Universal Robots URScript: dusan_v3_nosensor.task.script

def dusan_v3_nosensor():
  # Preamble Script.
  # Test Preamble Script To Be Added In The Future.
  set_safety_mode_transition_hardness(1)
  # Configuration Preamble Script.
  # Configuration variables.
  #
  global Home_joint
  Home_joint = [0.55498, -1.00739, -2.64993, -1.05507, 1.5708, 0.55497]
  #
  global Home_pose
  Home_pose = [0.33684, -0.00001, 0.31805, 3.14159, 0, -1.57079]
  # 시작 포즈 (입력레지스터 316~321). UI가 저장한 값
  global start_pose
  start_pose = [0.33684, -0.00001, 0.31805, 3.14159, 0, -1.57079]
  # 0=이 변수값 사용, 1=Modbus 310~321 사용 (레지스터 308)
  global pose_src
  pose_src = 0
  # 작업 속도 입력 [mm/s] (입력레지스터 306). 0이면 v_l 유지
  global spd_in
  spd_in = 0
  # 로봇 자체 속도 비율 [%] 2~100 (입력레지스터 307)
  global spd_ratio
  spd_ratio = 100
  # 0=이 변수값 사용, 1=Modbus 256~259 사용 (레지스터 266)
  global param_src
  param_src = 0
  # 중앙 접촉 센서 1차 — ON 이면 적정 눌림 위치
  global di_touch
  di_touch = 0
  # 중앙 접촉 센서 2차 — ON 이면 눌림 한계. TCP +Y 로 후퇴한다
  global di_limit
  di_limit = 1
  # 도면 반지름(안쪽 면) [mm]. 레지스터 260 을 0.1mm 로 받고, dus_init 이 두께를 더해 훑는 면 반지름으로 바꾼다
  global app_radius
  app_radius = 894.59998
  # 제품 두께 [mm]. 레지스터 261 을 0.1mm 단위로 받는다. UT 기록용
  global app_thick
  app_thick = 10
  # 격자 가로 = 호 길이 [mm] (레지스터 256). 로봇이 실제로 지나는 거리. 현이 아니다
  global app_arc
  app_arc = 1110
  # EOAT 가로(호 방향) [mm]. 레지스터 262. 5축 X형 257 / 8축 직사각 186
  global eoat_w
  eoat_w = 257
  # EOAT 세로 [mm]. 레지스터 263. 5축 257 / 8축 316(세로로 길게). 스캐너 밴드 높이로 쓴다
  global eoat_h
  eoat_h = 257
  # TCP 가 실제로 움직일 호 길이 [mm] = app_arc - eoat_w. dus_init 이 계산
  global arc_run
  arc_run = 853
  # 곡률 중심 X [m]. probe_l 이 계산
  global arc_ox
  arc_ox = 1.53144
  # 곡률 중심 Y [m]. probe_l 이 계산
  global arc_oy
  arc_oy = -0.00002
  # 원점(zero_pose)이 곡률 중심에서 보이는 각 [rad]
  global arc_phi0
  arc_phi0 = 2.66484
  # 호 기준이 잡혔는지. True 여야 호 위치를 발행한다
  global arc_ok
  arc_ok = True
  # 원점부터 지금까지의 호 위 거리 [mm]. 레지스터 286 으로 발행
  global arc_s
  arc_s = 0
  # 호 반각 [rad] = app_arc/(2*app_radius). dus_init 이 계산
  global arc_half
  arc_half = 0.47675
  # 센서로 잰 적정 눌림 보정량 [m]. 계산한 3점을 TCP -Y 로 이만큼 더 민다
  global press_off
  press_off = 0
  # 자세 보정 중 한 걸음 전진/후퇴 거리 [mm]
  global seek_step
  seek_step = 2
  # 전진·회전 되풀이 최대 횟수. 넘으면 포기하고 진행
  global seek_tries
  seek_tries = 80
  # 전진 최대 거리 [mm]. 센서가 없으면 여기까지 가고 멈춘다
  global seek_limit
  seek_limit = 400
  # 센서판: 계산한 좌우 끝점 접근 전 대기 거리 [mm](TCP +Y로 물러난 지점). 논센서판: 센서 없이 전진할 고정 거리 [mm]
  global probe_dist
  probe_dist = 300
  # [임시판 전용] 중앙이 가장자리보다 더 전진할 거리 [mm]. 0 이면 app_diameter 로 자동 계산(바깥 볼록면이라 음수가 나온다). 손으로 넣으려면 0 이 아닌 값을 준다
  global probe_bow
  probe_bow = 0
  # [임시판 전용] 원통 지름 [mm]. probe_bow 가 0 일 때 호의 볼록량을 이 값으로 계산한다 (센서가 붙으면 필요 없다)
  global app_diameter
  app_diameter = 1669
  # 측정 후 후퇴 거리 [mm]
  global back_off
  back_off = 100
  # 가로 패스를 나누는 구간 길이 [mm]. 작을수록 X 보정이 촘촘하다
  global seg_len
  seg_len = 50
  # movel(스캔 제외) 속도 [m/s]. dus_init 이 150mm/s 로 상한을 자른다
  global v_l
  v_l = 0.15
  # movel(스캔 제외) 가속도 [m/s^2]. 필요하면 각 스크립트가 그 자리에서 바꿔 쓴다
  global a_l
  a_l = 1.2
  # movej 속도 [rad/s] (20 deg/s). dus_init 이 0.50 rad/s 로 상한을 자른다 — 조그 상한과 같다. 펜던트 MoveJ 노드(홈 복귀)는 이 값을 직접 참조하지 못하므로 노드 쪽 수치도 같이 맞춰 둬야 한다
  global v_j
  v_j = 0.3490658503988659
  # movej 가속도 [rad/s^2] (40 deg/s^2)
  global a_j
  a_j = 0.698131700835289
  # 스캔 movel/movec 속도 [m/s]. 고정 스펙 100mm/s
  global v_scan
  v_scan = 0.1
  # 스캔 movel/movec 가속도 [m/s^2]. 고정 스펙 400mm/s^2
  global a_scan
  a_scan = 0.4
  # 작업 영역 좌우 너비 [mm] (입력레지스터 256)
  global app_width
  app_width = 821.05219
  # 작업 영역 높이 [mm] (입력레지스터 257)
  global app_height
  app_height = 500
  # 스캐너 세로 유효높이 [mm] (입력레지스터 258)
  global scan_h
  scan_h = 257
  # 세로 겹침 [mm] (입력레지스터 259)
  global overlap
  overlap = 20
  # 상승 피치 = scan_h - overlap [mm] (고정)
  global pitch
  pitch = 237
  # 가로 패스 수
  global rows
  rows = 3
  # 완료한 가로 패스 수
  global row_idx
  row_idx = 1
  # 1=오른쪽(Y-) 차례, -1=왼쪽(Y+) 차례
  global dir_sign
  dir_sign = -1
  #
  global pass_done
  pass_done = 0
  # 측정 완료한 점 수 (0~3)
  global n_probe
  n_probe = 3
  # 센서로 검출된 점 수
  global n_hit
  n_hit = 0
  # 중앙 측정 X [m]
  global p_cx
  p_cx = 0.63684
  # Y+ 끝 측정 X [m]
  global p_lx
  p_lx = 0.7366
  # Y- 끝 측정 X [m]
  global p_rx
  p_rx = 0.7366
  # 중앙 Y [m]
  global y_c
  y_c = -0.00001
  #
  global y_l
  y_l = 0.30185
  #
  global y_r
  y_r = -0.29815
  # 너비의 절반 [m]
  global half
  half = 0.3
  # 벽면 2차식 계수 : x = qa*dy^2 + qb*dy + qc, dy = Y - y_c
  global qa
  qa = 0
  # 벽면 2차식 1차항
  global qb
  qb = 0
  # 벽면 2차식 상수항 (= 중앙 X)
  global qc
  qc = 0
  #
  global zero_ok
  zero_ok = True
  #
  global x_start
  x_start = [0.33684, -0.00001, 0.32105, 3.14159, -0, -1.57079]
  #
  global z_base
  z_base = 0.32105
  # 원점 = Y+ 끝 측정 위치
  global zero_pose
  zero_pose = [0.7366, 0.41051, 0.32105, 3.14159, -0.00001, -2.04755]
  # pose_inv(zero_pose)
  global zero_inv
  zero_inv = [0.70276, 0.46608, 0.32105, -3.14159, 0, -2.04755]
  # 현재 절대 TCP (260~265 로 발행)
  global cur_pose
  cur_pose = [0.7236, -0.38435, 0.55805, 3.14159, -0.00001, -1.12675]
  # 원점 기준 상대 pose (280~285 로 발행)
  global rel_pose
  rel_pose = [-0.013, -0.79486, 0.237, -0, -0, 0.9208]
  # 현재 구간 목표 pose
  global tgt_pose
  tgt_pose = [0.7366, -0.41054, 0.55805, -3.14159, -0.00001, -1.09406]
  #
  global dy
  dy = 0.3
  #
  global y_from
  y_from = -0.30001
  #
  global y_to
  y_to = 0.29999
  #
  global n_seg
  n_seg = 12
  #
  global i_seg
  i_seg = 13
  # 누적 이동거리 [mm]
  global path_len
  path_len = 1090
  # 워치독 카운터
  global alive
  alive = 14011
  # 이동 스레드 핸들
  global mv_h
  mv_h = 0
  # 발행 스레드 핸들
  global pub_h
  pub_h = 855631424
  # 정렬 전 기준 자세. 측정점 사이를 이동할 때 여기로 되돌린다 (probe_c 가 채운다)
  global probe_rot
  probe_rot = [0.33684, -0.00001, 0.31805, 3.14159, 0, -1.57079]
  # movec 의 mode. 0 = 자세 고정
  global arc_mode
  arc_mode = 0
  # 중앙 측정 pose — movec 의 경유점 (330~335 로 발행)
  global p_c_pose
  p_c_pose = [0.63684, -0.00001, 0.32105, 3.14159, -0.00001, -1.5708]
  # Y- 끝 측정 pose — movec 의 도착점 (340~345 로 발행)
  global p_r_pose
  p_r_pose = [0.7366, -0.41054, 0.32105, 3.14159, -0.00001, -1.09405]
  # movec 경유점 (현재 높이로 갈아끼운 것)
  global via_pose
  via_pose = [0.63684, -0.00001, 0.55805, 3.14159, -0.00001, -1.5708]
  # movec 도착점 (현재 높이로 갈아끼운 것)
  global to_pose
  to_pose = [0.7366, 0.41051, 0.55805, 3.14159, -0.00001, -2.04755]
  # 가로 패스 시작 시점의 Z [m]
  global z_now
  z_now = 0.55805
  set_tool_analog_io_work_mode(3)
  set_tool_digital_io_work_mode(0)
  set_tool_analog_input_domain(0)
  set_tool_analog_output_domain(0)
  set_tool_digital_io_config(0,0,False,False)
  set_tool_digital_io_config(1,0,False,False)
  set_tool_digital_io_config(2,0,False,False)
  set_tool_digital_io_config(3,0,False,False)
  tool_serial_config(False,115200,0,1,modbus_rtu = False,usage = 0)
  set_tool_voltage(0)
  set_tcp([0.0, 0.0, 0.0, 0.0, 0.0, 0.0])
  set_payload(0.0, [0.0, 0.0, 0.0], [0.0, 0.0, 0.0, 0.0, 0.0, 0.0])
  set_standard_analog_input_domain(0, 1)
  set_standard_analog_input_domain(1, 1)
  set_standard_analog_output_domain(0, 0)
  set_standard_analog_output_domain(1, 0)
  set_input_actions_to_default()
  set_gravity([0.0, 0.0, 9.82])
  # Frame variables.
  # Temporary frame variables.
  # Conveyor Config
  #--------------- lifting Column Function -----------------
  liftingColumn = rpc_factory("xmlrpc","http://0.0.0.0:9120/RPC2")
  def visualLimitLiftingColumn(visualMinLimit=0, visualMaxLimit=500):
      # 设置升降柱虚拟限位
      # visualMinLimit:虚拟最低限位
      # visualMaxLimit:虚拟最高限位
      liftingColumn.setVisualLimit(visualMinLimit, visualMaxLimit)
  def liftingCurrentHeight():
      # 获取升降柱当前高度
      return liftingColumn.currentHeight()
  def liftingStop():
      # 停止升降柱移动
      return liftingColumn.stop()
  def getLiftingTravel():
      # 获取升降柱总行程
      return 500
  def getLiftingMinLimit():
      # 获取升降柱最低限位
      return 0
  def getLiftingMaxLimit():
      # 获取升降柱最高限位
      return 500
  def connectLiftingColumn(ip, port=502, slaveID=1,length=500):
      # 链接升降柱
      # ip:升降柱ip
      # port:升降柱端口号
      # slaveID:从站ID
      # length:升降柱总行程
      liftingColumn.setLiftingLength(length)
      return liftingColumn.connect(ip, port, slaveID)
  def disConnectLiftingColumn():
      # 断开升降柱链接
      return liftingColumn.disConnect()
  def moveLiftingColumn(pos, speed, block=True):
      # 升降柱移动命令
      # pos: 升降柱位置
      # speed: 升降柱速度
      if pos > liftingColumn.getMaxLimit():
          popup(s="Move pos is over limit max.", title="LiftingColumnAdapter Plugin Error", blocking=True)
          halt()
      moveRes = liftingColumn.move(pos, speed)
      if not moveRes:
          popup("Lifting Column Failed To Move! Please Check Lifting Column Status!", title="LiftingColumnAdapter Plugin Error", error=True, blocking=True)
      while block:
          currentHeight = liftingColumn.currentHeight()
          errorCode = liftingColumn.errorCode()
          if currentHeight < pos + 2 and currentHeight > pos - 2 and currentHeight != -1:
              liftingColumn.clearMovingFlag()
              return True
          if errorCode > 0:
              liftingColumn.stop()
              liftingColumn.clearMovingFlag()
              popup(s="Lifting error ,stop task.Error code: " + str(errorCode), title="LiftingColumnAdapter Plugin Error", blocking=True)
              halt()
              return False
          sleep(0.2)
      return moveRes
  #--------------- lifting Column Function -----------------
  # Set Node Preamble Script.
  # Loop Node Preamble Script.
  # Waypoint Node Preamble Script.
  # Initial Variables value.
  global Loop_1
  def calculate_point_to_move_towards(frame, direction, position_distance):
    posDir = [direction[0], direction[1], direction[2]]
    if (norm(posDir) < 1e-6):
      return get_target_waypoint()
    end
    direction_vector_normalized = normalize(posDir)
    displacement_pose = [direction_vector_normalized[0] * position_distance,direction_vector_normalized[1] * position_distance,direction_vector_normalized[2] * position_distance,0,0,0]
    wanted_displacement_in_base_frame = pose_sub(pose_trans(frame, displacement_pose), frame)
    return pose_add(get_target_waypoint(), wanted_displacement_in_base_frame)
  end
  # Timer Node Preamble Script.
  # SubTask Node Preamble Script.
  # Before Start Preamble Script.
  # Thread Node Preamble Script.
  # Event Node Preamble Script.
  # Main Task Script.
  while (True):
    $ LINE: (2, "로봇 메인 작업")
    $ LINE: (3, "1 [스크립트파일] dus_init.script")
    $ LINE: (4, "스크립트")
    # =============================================================================
    #  dus_init.script — dusan_v3
    #  파라미터를 읽고 피치·행수를 계산한다. 실시간 발행 스레드를 띄운다
    #
    #  펜던트에서 "1_init" 자리에 스크립트 노드를 파일(File) 모드로 넣고 지정한다.
    #
    #  ※ def main() 으로 감싸지 말 것 (펜던트가 호출하지 않는다)
    #  ※ 최상위에 global 을 쓰지 말 것 (preamble 이 이미 선언·대입해 뒀다)
    #  ※ if / while 은 반드시 end 로 닫을 것
    # =============================================================================

    def ini_w1(a, v):
      if (v > 32000):
        v = 32000
      end
      if (v < -32000):
        v = -32000
      end
      write_port_register(a, floor(v + 0.5))
    end


    # 로봇 자체 레지스터 384~389 와 같은 단위.  길이 0.1mm, 회전 mRad
    def ini_w6(a, p):
      ini_w1(a, p[0] * 10000)
      ini_w1(a + 1, p[1] * 10000)
      ini_w1(a + 2, p[2] * 10000)
      ini_w1(a + 3, p[3] * 1000)
      ini_w1(a + 4, p[4] * 1000)
      ini_w1(a + 5, p[5] * 1000)
    end


    # 절대 TCP(260~265) 는 항상 발행한다. 원점기준 상대좌표(280~285)와 호
    # 위치(286/287)는 원점(zero_pose)이 잡혀 있으면(zero_ok/arc_ok) 항상
    # 내보낸다 — TPAC 의 "Plane" 이 실제 TCP 이동거리를 보여줘야 하므로 ㄹ자
    # 스캔 중(state=4)만이 아니라 3점측정 후 원점복귀·다음 줄 이동 중에도
    # 값이 살아 있어야 한다. 원점이 아직 없으면(zero_ok==False) [0,0,0,0,0,0]
    # 을 쏜다.
    #
    # 위치는 베이스 좌표계 그대로 빼서 쓴다(cur - zero). 원래는
    # pose_trans(zero_inv, cur_pose)로 툴 좌표계 기준값을 냈는데, 툴이
    # 벽을 비스듬히 보고 있으면 베이스 Z+ 로 올라가도 이 값의 Z 성분이
    # 음수로 커지는 문제가 있었다. register_map.txt 4항의 역변환 공식
    # base = R_zero * rel_tcp 은 rel_tcp = R_zero^T * (cur-zero) 이므로
    # 결국 cur - zero 와 정확히 같다(회전행렬을 걸었다 다시 푸는 셈).
    # 그러니 처음부터 베이스 좌표계로 빼면 회전행렬 없이 같은 결과이고,
    # 세로(Z)가 위로 갈수록 커지도록 직관과도 맞는다.
    def pub_rel():
      global cur_pose
      global rel_pose
      global alive
      cur_pose = get_actual_tcp_pose()
      ini_w6(260, cur_pose)
      if (zero_ok == True):
        rel_pose = [cur_pose[0] - zero_pose[0],
              cur_pose[1] - zero_pose[1],
              cur_pose[2] - zero_pose[2],
              cur_pose[3] - zero_pose[3],
              cur_pose[4] - zero_pose[4],
              cur_pose[5] - zero_pose[5]]
        ini_w6(280, rel_pose)
      else:
        ini_w6(280, [0, 0, 0, 0, 0, 0])
      end
      # ---- 호 위 위치 (TPAC 스캔 축) ----------------------------------
      # 좌표를 그대로 주면 현(1031.8)으로 7% 눌리고 호 위치에 비례하지도
      # 않는다. 원점부터 호를 따라 실제로 지난 거리를 계산해서 내보낸다.
      #   286 = 이번 줄의 호 위 거리 [0.1mm]  (0 ~ 11100)
      #   287 = 완료된 줄까지 더한 누적 [mm]
      if (arc_ok == True):
        adx = cur_pose[0] - arc_ox
        ady = cur_pose[1] - arc_oy
        aph = atan2(ady, adx) - arc_phi0
        # atan2 는 ±pi 로 감기므로 한 바퀴 보정한다
        if (aph > 3.14159265):
          aph = aph - 6.28318531
        end
        if (aph < -3.14159265):
          aph = aph + 6.28318531
        end
        if (aph < 0):
          aph = -aph
        end
        arc_s = aph * app_radius
        ini_w1(286, arc_s * 10)
        ini_w1(287, path_len + arc_s)
      else:
        arc_s = 0
        ini_w1(286, 0)
        ini_w1(287, path_len)
      end

      alive = alive + 1
      if (alive > 30000):
        alive = 0
      end
      write_port_register(293, alive)
    end


    # 제어주기마다 도는 발행 스레드. 이 뒤로는 평범한 movel 을 써도
    # 이동 중 좌표가 계속 나간다.
    def pub_thread():
      while (True):
        pub_rel()
        sync()
      end
    end


    # ------------------------------------------------------------------ 본문
    # 266 = 1 이면 외부(Modbus)가 준 값을, 0 이면 펜던트 변수값을 쓴다
    #   256 호 길이 [mm]   257 격자 높이 [mm]   258 스캐너 높이 [mm]
    #   259 겹침 [mm]      260 반지름 [0.1mm]   261 두께 [0.1mm]
    # 260/261 만 0.1mm 인 이유: 반지름이 834.6 처럼 소수라 정수 mm 로는
    # 호 모양이 눈에 띄게 틀어진다.
    if (read_port_register(266, True) == 1):
      app_arc = read_port_register(256, True)
      app_height = read_port_register(257, True)
      scan_h = read_port_register(258, True)
      overlap = read_port_register(259, True)
      app_radius = read_port_register(260, True) * 0.1
      app_thick = read_port_register(261, True) * 0.1
      eoat_w = read_port_register(262, True)
      eoat_h = read_port_register(263, True)
    end

    # ---- EOAT(검사 프로브 뭉치) 크기 ------------------------------------------
    # 프로브가 EOAT 폭만큼 퍼져 있으므로 TCP 가 격자 끝까지 갈 필요가 없다.
    # 양 끝에서 EOAT 의 **반**씩 안쪽으로 들어가면 프로브 가장자리가 끝에 닿는다.
    # 그래서 실제 이동 호 길이는 덮는 길이에서 EOAT 폭 하나를 뺀 값이다.
    #   5축 X형 257x257 -> 1110-257 = 853,  8축 186x316 -> 1110-186 = 924
    # 세로도 마찬가지로 EOAT 세로가 곧 한 줄이 덮는 밴드 높이(scan_h)가 된다.
    if (eoat_h > 0):
      scan_h = eoat_h
    end
    if (eoat_w > 0):
      arc_run = app_arc - eoat_w
      if (arc_run < 1):
        # EOAT 가 격자보다 넓다 = 한 자리에서 다 덮는다. 움직이지 않는다.
        arc_run = 0
      end
    else:
      arc_run = app_arc
    end

    if (app_arc <= 0):
      app_arc = 1000
    end
    if (app_radius < 0):
      app_radius = 0
    end

    # ---- 훑는 면의 반지름 -----------------------------------------------------
    # 도면 반지름은 안쪽(오목) 면 기준이고 로봇은 바깥(볼록) 면을 훑으므로
    # 두께를 더해야 실제로 손이 닿는 면의 반지름이 된다 (834.6 + 10 = 844.6).
    if (app_radius > 0):
      app_radius = app_radius + app_thick
    end

    # ---- 호 기하 --------------------------------------------------------------
    # 받은 값은 **호 길이**다(현이 아니다). 반각 t = L/(2R), 현 c = 2R*sin(t).
    #   시험 벽: L=1110, R=844.6 -> t=0.6571 rad(37.6deg), c=1031.8
    # 로봇이 실제로 지나는 길이는 movec 가 호를 따라가므로 호 길이(1110) 다.
    if (app_radius > 0):
      arc_half = arc_run / (2.0 * app_radius)
      app_width = 2.0 * app_radius * sin(arc_half)
    else:
      arc_half = 0
      app_width = arc_run
    end

    if (app_height < 0):
      app_height = 0
    end
    if (scan_h <= 0):
      scan_h = 200
    end
    if (overlap < 0):
      overlap = 0
    end
    if (overlap >= scan_h):
      overlap = scan_h - 10
    end

    # ---- 속도/가속도 : 전역 변수로 관리한다 ----------------------------------
    #   movel(스캔 제외)       : a_l, v_l
    #   movej(홈 복귀 등)      : a_j, v_j
    #   스캔 movel/movec       : a_scan, v_scan  (고정 스펙 100 mm/s / 400 mm/s^2)
    # 필요하면 각 스크립트가 그 자리에서 값을 바꿔 써도 된다 — 예를 들어
    # 접촉 위치 진입처럼 더 천천히 움직여야 할 때는 v_l 을 따로 두지 않고
    # `v_l / 3.0` 처럼 그 movel 호출 하나에만 적용한다(전역값 자체는 안 바뀜).
    #
    # 안전 규정: 스캔 외 동작은 150 mm/s 를 넘으면 안 된다. 관절 이동의
    # 각속도도 여기에 맞춰 조그와 같은 상한(0.50 rad/s)을 넘지 않게 자른다.
    # 306 = 작업 속도 [mm/s]. v_l 로 쓴다. 0 이면 변수값을 유지한다.
    # 307 = 로봇 자체 속도 비율 [%] 2~100. 모든 이송 속도에 곱한다.
    spd_in = read_port_register(306, True)
    if (spd_in > 0):
      v_l = spd_in / 1000.0
    end

    # ---- 안전 상한 : 비율(307)을 곱하기 전에 자르므로 100 % 가 곧 이 값이다 --
    v_l_limit = 0.150
    if (v_l > v_l_limit):
      v_l = v_l_limit
    end
    v_j_limit = 0.50
    if (v_j > v_j_limit):
      v_j = v_j_limit
    end

    spd_ratio = read_port_register(307, True)
    if (spd_ratio < 2):
      spd_ratio = 100
    end
    if (spd_ratio > 100):
      spd_ratio = 100
    end
    v_l = v_l * spd_ratio / 100.0
    v_j = v_j * spd_ratio / 100.0
    v_scan = v_scan * spd_ratio / 100.0

    # ---- 기준 위치 : 308 이 1 이면 310~321 의 값을 쓴다 --------------------
    # 310~315 홈 관절값 [mRad], 316~321 시작 pose (길이 0.1mm, 회전 mRad)
    if (read_port_register(308, True) == 1):
      Home_joint = [read_port_register(310, True) / 1000.0,
             read_port_register(311, True) / 1000.0,
             read_port_register(312, True) / 1000.0,
             read_port_register(313, True) / 1000.0,
             read_port_register(314, True) / 1000.0,
             read_port_register(315, True) / 1000.0]
      start_pose = [read_port_register(316, True) / 10000.0,
             read_port_register(317, True) / 10000.0,
             read_port_register(318, True) / 10000.0,
             read_port_register(319, True) / 1000.0,
             read_port_register(320, True) / 1000.0,
             read_port_register(321, True) / 1000.0]
      Home_pose = get_forward_kin(Home_joint)
    end

    # 상승 피치 = 스캐너 높이 - 겹침 (고정)
    pitch = scan_h - overlap
    if (pitch <= 0):
      pitch = 10
    end

    # 스캐너가 한 자리에서 scan_h 를 훑으므로
    # 마지막 패스가 (높이 - scan_h) 이상이면 사각형 전체가 덮인다
    rows = ceil((app_height - scan_h) * 1.0 / pitch) + 1
    if (rows < 1):
      rows = 1
    end
    if (rows > 200):
      popup(s = "ROWS OVER LIMIT(200). CHECK HEIGHT/SCAN_H/OVERLAP", title = "dusan_v3", blocking = True)
      write_port_register(290, 9)
      halt()
    end

    row_idx = 0
    dir_sign = 1
    pass_done = 0
    path_len = 0
    alive = 0
    zero_ok = False
    n_probe = 0
    n_hit = 0
    qa = 0
    qb = 0
    qc = 0

    write_port_register(290, 0)
    write_port_register(291, 0)
    write_port_register(292, rows)
    write_port_register(293, 0)
    write_port_register(294, 0)
    write_port_register(295, 0)
    write_port_register(296, pitch)
    write_port_register(297, 0)
    write_port_register(298, 0)
    write_port_register(299, 0)  # probe_error: 0=정상, 1/2/3=probe_c/l/r 접촉 실패
    write_port_register(304, 0)
    write_port_register(305, 0)

    # 실시간 발행 스레드 기동
    pub_h = start_thread(pub_thread, (), detach_mode = True)
    $ LINE: (5, "2 move_home")
    $ LINE: (6, "If")
    if (get_actual_tcp_pose()[2]<Home_pose[2]-0.001):
      $ LINE: (7, "MoveL")
      $ LINE: (8, "방향 로봇 Z+")
      global move_thread_flag_8
      move_thread_flag_8 = 0
      def move_thread_8():
        global move_thread_flag_8
        move_thread_flag_8 = 1
        towardsPos = calculate_point_to_move_towards([0.0, 0.0, 0.0, 0.0, 0.0, 0.0], [0.0,0.0,1.0], 1000.0)
        movel(towardsPos, a=0.6, v=0.15)
        move_thread_flag_8 = 2
      end
      move_thread_flag_8 = 0
      move_thread_han_8 = start_thread(move_thread_8, (), detach_mode = False)
      while (True):
        if (get_actual_tcp_pose()[2]>=Home_pose[2]-0.001):
          stop_thread(move_thread_han_8)
          stopl(0.6)
          $ LINE: (9, "Until (표현식)")
          break
        end
        sync()
      end
    end
    $ LINE: (10, "MoveJ")
    $ LINE: (11, "Home_joint", "after")
    movej(Home_joint, a=0.698131700835289, v=0.3490658503988659)
    $ LINE: (12, "3 [스크립트파일] dus_probe_c.script")
    $ LINE: (13, "스크립트")
    # =============================================================================
    #  dus_probe_c.script — dusan_v3
    #  중앙에서 전진해 벽을 찾고 pose 를 기록한 뒤 후퇴한다
    #
    #  펜던트에서 "3_probe_center" 자리에 스크립트 노드를 파일(File) 모드로 넣고 지정한다.
    #
    #  ※ def main() 으로 감싸지 말 것 (펜던트가 호출하지 않는다)
    #  ※ 최상위에 global 을 쓰지 말 것 (preamble 이 이미 선언·대입해 뒀다)
    #  ※ if / while 은 반드시 end 로 닫을 것
    # =============================================================================

    def pc_w1(a, v):
      if (v > 32000):
        v = 32000
      end
      if (v < -32000):
        v = -32000
      end
      write_port_register(a, floor(v + 0.5))
    end


    # 로봇 자체 레지스터 384~389 와 같은 단위.  길이 0.1mm, 회전 mRad
    def pc_w6(a, p):
      pc_w1(a, p[0] * 10000)
      pc_w1(a + 1, p[1] * 10000)
      pc_w1(a + 2, p[2] * 10000)
      pc_w1(a + 3, p[3] * 1000)
      pc_w1(a + 4, p[4] * 1000)
      pc_w1(a + 5, p[5] * 1000)
    end

    write_port_register(290, 2)
    y_c = get_actual_tcp_pose()[1]
    z_base = get_actual_tcp_pose()[2]

    # 정렬 기준 자세 : 측정점 사이를 이동할 때(probe_l/r, goto_zero) 이 회전으로
    # 되돌아온다. 움직이기 전에 남겨 둔다 (센서판 probe_c 와 같은 역할).
    x_start = get_actual_tcp_pose()
    probe_rot = x_start

    # 중앙점 접근  [임시판 : 센서가 없으니 정해진 거리만 전진]
    # 센서판과 달리 눌림을 못 재므로 probe_dist 를 그대로 믿는다.
    # 전진은 TCP -Y (호를 그리며 손 방향이 바뀌므로 베이스 기준이면 안 된다).
    movel(pose_trans(x_start, [0, -probe_dist * 0.001, 0, 0, 0, 0]),
          a = a_l, v = v_l / 3.0)  # 접촉 위치 진입: 천천히

    n_probe = n_probe + 1
    write_port_register(304, n_probe)
    write_port_register(305, n_hit)

    # movec 의 경유점으로 쓸 pose 전체를 남긴다
    p_c_pose = get_actual_tcp_pose()
    p_cx = p_c_pose[0]
    write_port_register(300, floor(p_cx * 10000 + 0.5))
    pc_w6(330, p_c_pose)

    # 벽에서 물러난다 (온 만큼 그대로 되돌아간다)
    movel(x_start, a = a_l, v = v_l)
    $ LINE: (14, "2 move_home")
    $ LINE: (15, "If")
    if (get_actual_tcp_pose()[2]<Home_pose[2]-0.001):
      $ LINE: (16, "MoveL")
      $ LINE: (17, "방향 로봇 Z+")
      global move_thread_flag_17
      move_thread_flag_17 = 0
      def move_thread_17():
        global move_thread_flag_17
        move_thread_flag_17 = 1
        towardsPos = calculate_point_to_move_towards([0.0, 0.0, 0.0, 0.0, 0.0, 0.0], [0.0,0.0,1.0], 1000.0)
        movel(towardsPos, a=0.6, v=0.15)
        move_thread_flag_17 = 2
      end
      move_thread_flag_17 = 0
      move_thread_han_17 = start_thread(move_thread_17, (), detach_mode = False)
      while (True):
        if (get_actual_tcp_pose()[2]>=Home_pose[2]-0.001):
          stop_thread(move_thread_han_17)
          stopl(0.6)
          $ LINE: (18, "Until (표현식)")
          break
        end
        sync()
      end
    end
    $ LINE: (19, "MoveJ")
    $ LINE: (20, "Home_joint", "after")
    movej(Home_joint, a=0.698131700835289, v=0.3490658503988659)
    $ LINE: (21, "4 [스크립트파일] dus_probe_l.script")
    $ LINE: (22, "스크립트")
    # =============================================================================
    #  dus_probe_l.script — dusan_v3
    #  Y- 로 너비/2 이동해 측정한다. 이 점이 원점이 된다
    #
    #  펜던트에서 "4_probe_left" 자리에 스크립트 노드를 파일(File) 모드로 넣고 지정한다.
    #
    #  ※ def main() 으로 감싸지 말 것 (펜던트가 호출하지 않는다)
    #  ※ 최상위에 global 을 쓰지 말 것 (preamble 이 이미 선언·대입해 뒀다)
    #  ※ if / while 은 반드시 end 로 닫을 것
    # =============================================================================


    def nl_arc(mid, th):
      # 중앙 접점 mid 에서 호를 따라 th [rad] 만큼 돌아간 점(자세 포함).
      # 센서판(dus_probe_l)과 같은 계산이다.
      #
      # 원통은 세워져 있으므로 호는 **수평면** 안에 있다. 그래서
      #   (1) 곡률 중심 O 는 접점에서 '전진 방향(TCP -Y)의 **수평 성분**'으로 R.
      #   (2) 회전은 O 를 지나는 **수직축(베이스 Z)** 으로 한다.
      #       툴 로컬 Z 로 돌리면 호가 수평면을 벗어나 현이 짧아진다.
      # 자세도 같이 돌아가므로 각 점에서 손이 그 자리의 법선을 본다.
      if (app_radius <= 0):
        return mid
      end
      fwd = pose_trans(mid, [0, -1.0, 0, 0, 0, 0])
      dx = fwd[0] - mid[0]
      dy = fwd[1] - mid[1]
      n = sqrt(dx * dx + dy * dy)
      if (n < 0.0001):
        return mid
      end
      r = app_radius * 0.001
      o_t = [mid[0] + dx / n * r, mid[1] + dy / n * r, 0, 0, 0, 0]
      return pose_trans(o_t, pose_trans([0, 0, 0, 0, 0, th], pose_trans(pose_inv(o_t), mid)))
    end


    write_port_register(290, 3)

    # 양 끝을 계산해 베이스 Y 가 작은 쪽을 Y-(원점), 큰 쪽을 Y+ 로 나눈다.
    # 손이 어느 방향을 보느냐에 따라 +t 가 어느 쪽으로 갈지 달라지므로
    # 부호를 미리 못 박지 않고 실제 좌표로 가른다.
    end_a = nl_arc(p_c_pose, arc_half)
    end_b = nl_arc(p_c_pose, -arc_half)
    if (end_a[1] <= end_b[1]):
      zero_pose = end_a
      p_r_pose = end_b
    else:
      zero_pose = end_b
      p_r_pose = end_a
    end

    # 이 자리가 원점이자 movec 의 시작점이다 (회전값 포함)
    p_lx = zero_pose[0]
    write_port_register(301, floor(p_lx * 10000 + 0.5))
    zero_inv = pose_inv(zero_pose)
    zero_ok = True

    # ---- 호 위 위치를 실시간으로 내보내기 위한 기준 ---------------------------
    # TPAC 은 스캔 축 위치로 **호 길이**를 받아야 한다. 좌표를 그대로 주면
    # 현(1031.8)으로 7% 눌리고, 게다가 호 위치에 비례하지 않아 1/4·3/4 지점에서
    # 14.6mm 씩 어긋난다(C-scan 이 앞뒤로 밀려 찍힌다).
    # 곡률 중심과 원점의 방위각을 남겨 두면, 발행 스레드가 매 주기
    #   s = R * |현재각 - 원점각|
    # 으로 호 위 실제 거리를 계산할 수 있다.
    if (app_radius > 0):
      fwd0 = pose_trans(p_c_pose, [0, -1.0, 0, 0, 0, 0])
      d0x = fwd0[0] - p_c_pose[0]
      d0y = fwd0[1] - p_c_pose[1]
      n0 = sqrt(d0x * d0x + d0y * d0y)
      if (n0 > 0.0001):
        arc_ox = p_c_pose[0] + d0x / n0 * app_radius * 0.001
        arc_oy = p_c_pose[1] + d0y / n0 * app_radius * 0.001
        arc_phi0 = atan2(zero_pose[1] - arc_oy, zero_pose[0] - arc_ox)
        arc_ok = True
      end
    end

    # 회전각이 다른 채로 벽 쪽 목표로 바로 가면 볼록한 곡면을 가로질러
    # 충돌한다. 목표 자세(zero_pose 의 회전) 그대로 뒤로 물러난 지점까지
    # 먼저 이동한 뒤, 그 자세로 곧장 전진해 들어간다.
    l_stand = pose_trans(zero_pose, [0, probe_dist * 0.001, 0, 0, 0, 0])
    movel(l_stand, a = a_l, v = v_l)
    movel(zero_pose, a = a_l, v = v_l / 3.0)  # 접촉 위치 진입: 천천히

    n_probe = n_probe + 1
    write_port_register(304, n_probe)
    write_port_register(305, n_hit)

    # 다음 동작(probe_r)으로 넘어가기 전에 다시 물러난다
    movel(l_stand, a = a_l, v = v_l)
    $ LINE: (23, "2 move_home")
    $ LINE: (24, "If")
    if (get_actual_tcp_pose()[2]<Home_pose[2]-0.001):
      $ LINE: (25, "MoveL")
      $ LINE: (26, "방향 로봇 Z+")
      global move_thread_flag_26
      move_thread_flag_26 = 0
      def move_thread_26():
        global move_thread_flag_26
        move_thread_flag_26 = 1
        towardsPos = calculate_point_to_move_towards([0.0, 0.0, 0.0, 0.0, 0.0, 0.0], [0.0,0.0,1.0], 1000.0)
        movel(towardsPos, a=0.6, v=0.15)
        move_thread_flag_26 = 2
      end
      move_thread_flag_26 = 0
      move_thread_han_26 = start_thread(move_thread_26, (), detach_mode = False)
      while (True):
        if (get_actual_tcp_pose()[2]>=Home_pose[2]-0.001):
          stop_thread(move_thread_han_26)
          stopl(0.6)
          $ LINE: (27, "Until (표현식)")
          break
        end
        sync()
      end
    end
    $ LINE: (28, "MoveJ")
    $ LINE: (29, "Home_joint", "after")
    movej(Home_joint, a=0.698131700835289, v=0.3490658503988659)
    $ LINE: (30, "5 [스크립트파일] dus_probe_r.script")
    $ LINE: (31, "스크립트")
    # =============================================================================
    #  dus_probe_r.script — dusan_v3
    #  Y+ 끝으로 이동해 측정한다. 3점이 movec 의 시작/경유/도착이 된다
    #
    #  펜던트에서 "5_probe_right" 자리에 스크립트 노드를 파일(File) 모드로 넣고 지정한다.
    #
    #  ※ def main() 으로 감싸지 말 것 (펜던트가 호출하지 않는다)
    #  ※ 최상위에 global 을 쓰지 말 것 (preamble 이 이미 선언·대입해 뒀다)
    #  ※ if / while 은 반드시 end 로 닫을 것
    # =============================================================================

    def pr_w1(a, v):
      if (v > 32000):
        v = 32000
      end
      if (v < -32000):
        v = -32000
      end
      write_port_register(a, floor(v + 0.5))
    end


    # 로봇 자체 레지스터 384~389 와 같은 단위.  길이 0.1mm, 회전 mRad
    def pr_w6(a, p):
      pr_w1(a, p[0] * 10000)
      pr_w1(a + 1, p[1] * 10000)
      pr_w1(a + 2, p[2] * 10000)
      pr_w1(a + 3, p[3] * 1000)
      pr_w1(a + 4, p[4] * 1000)
      pr_w1(a + 5, p[5] * 1000)
    end


    p_rx = p_r_pose[0]
    write_port_register(302, floor(p_rx * 10000 + 0.5))
    pr_w6(340, p_r_pose)

    # probe_l 과 같은 이유로, 뒤로 물러난 지점을 거쳐 목표 자세 그대로 전진한다.
    r_stand = pose_trans(p_r_pose, [0, probe_dist * 0.001, 0, 0, 0, 0])
    movel(r_stand, a = a_l, v = v_l)
    movel(p_r_pose, a = a_l, v = v_l / 3.0)  # 접촉 위치 진입: 천천히

    n_probe = n_probe + 1
    write_port_register(304, n_probe)
    write_port_register(305, n_hit)

    # goto_zero 로 넘어가기 전에 다시 물러난다
    movel(r_stand, a = a_l, v = v_l)

    # 세 점이 그대로 movec 의 시작(원점) / 경유(중앙) / 도착(Y+ 끝) 이 된다.
    write_port_register(346, arc_mode)
    $ LINE: (32, "2 move_home")
    $ LINE: (33, "If")
    if (get_actual_tcp_pose()[2]<Home_pose[2]-0.001):
      $ LINE: (34, "MoveL")
      $ LINE: (35, "방향 로봇 Z+")
      global move_thread_flag_35
      move_thread_flag_35 = 0
      def move_thread_35():
        global move_thread_flag_35
        move_thread_flag_35 = 1
        towardsPos = calculate_point_to_move_towards([0.0, 0.0, 0.0, 0.0, 0.0, 0.0], [0.0,0.0,1.0], 1000.0)
        movel(towardsPos, a=0.6, v=0.15)
        move_thread_flag_35 = 2
      end
      move_thread_flag_35 = 0
      move_thread_han_35 = start_thread(move_thread_35, (), detach_mode = False)
      while (True):
        if (get_actual_tcp_pose()[2]>=Home_pose[2]-0.001):
          stop_thread(move_thread_han_35)
          stopl(0.6)
          $ LINE: (36, "Until (표현식)")
          break
        end
        sync()
      end
    end
    $ LINE: (37, "MoveJ")
    $ LINE: (38, "Home_joint", "after")
    movej(Home_joint, a=0.698131700835289, v=0.3490658503988659)
    $ LINE: (39, "6 [스크립트파일] dus_goto_zero.script")
    $ LINE: (40, "스크립트")
    # =============================================================================
    #  dus_goto_zero.script — dusan_v3
    #  측정이 끝난 뒤 원점(Y- 끝)으로 돌아가 스캔을 시작할 준비를 한다
    #
    #  펜던트에서 "6_goto_zero" 자리에 스크립트 노드를 파일(File) 모드로 넣고 지정한다.
    #
    #  ※ def main() 으로 감싸지 말 것 (펜던트가 호출하지 않는다)
    #  ※ 최상위에 global 을 쓰지 말 것 (preamble 이 이미 선언·대입해 뒀다)
    #  ※ if / while 은 반드시 end 로 닫을 것
    # =============================================================================

    def gz_w1(a, v):
      if (v > 32000):
        v = 32000
      end
      if (v < -32000):
        v = -32000
      end
      write_port_register(a, floor(v + 0.5))
    end


    def gz_w6(a, p):
      gz_w1(a, p[0] * 10000)
      gz_w1(a + 1, p[1] * 10000)
      gz_w1(a + 2, p[2] * 10000)
      gz_w1(a + 3, p[3] * 1000)
      gz_w1(a + 4, p[4] * 1000)
      gz_w1(a + 5, p[5] * 1000)
    end


    write_port_register(290, 3)

    # 현재 TCP 자세를 기준으로 가면 안 된다 — 직전 지점(p_r_pose)의 회전이
    # 그대로 남아 있어 zero_pose 의 회전과 다르고, 그 채로 위치만 옮기면
    # 볼록한 곡면을 가로질러 충돌한다. probe_l/r 과 같은 방식으로, zero_pose
    # 자세 그대로 뒤로 물러난 지점까지 먼저 이동한 뒤 그 자세로 전진해 들어간다.
    z_stand = pose_trans(zero_pose, [0, probe_dist * 0.001, 0, 0, 0, 0])
    movel(z_stand, a = a_l, v = v_l)
    movel(zero_pose, a = a_l, v = v_l / 3.0)  # 접촉 위치 진입: 천천히

    gz_w6(270, zero_pose)      # 원점 pose (스캔 중 변하지 않는다)
    write_port_register(294, 1)
    path_len = 0
    write_port_register(290, 4)
    $ LINE: (41, "루프 200 횟수")
    Loop_1 = 0
    while (Loop_1 < 200):
      $ LINE: (42, "스크립트")
      pass_done=0
      $ LINE: (43, "If")
      if (row_idx<rows and dir_sign>0 and pass_done==0):
        $ LINE: (44, "7 [스크립트파일] dus_pass_r.script")
        $ LINE: (45, "스크립트")
    # =============================================================================
    #  dus_pass_r.script — dusan_v3
    #  오른쪽(Y+) 으로 한 줄. 중앙을 경유점으로 하는 movec 원호
    #
    #  펜던트에서 "7_pass_right" 자리에 스크립트 노드를 파일(File) 모드로 넣고 지정한다.
    #
    #  ※ def main() 으로 감싸지 말 것 (펜던트가 호출하지 않는다)
    #  ※ 최상위에 global 을 쓰지 말 것 (preamble 이 이미 선언·대입해 뒀다)
    #  ※ if / while 은 반드시 end 로 닫을 것
    # =============================================================================

    def pr2_w1(a, v):
      if (v > 32000):
        v = 32000
      end
      if (v < -32000):
        v = -32000
      end
      write_port_register(a, floor(v + 0.5))
    end


    # 오른쪽(Y+) 으로 한 줄 — movec 원호 하나
    z_now = get_actual_tcp_pose()[2]
    via_pose = p_c_pose.copy()
    via_pose[2] = z_now
    to_pose = p_r_pose.copy()
    to_pose[2] = z_now
    movec(via_pose, to_pose, a = a_scan, v = v_scan, r = 0, mode = 1)

    row_idx = row_idx + 1
    dir_sign = -1
    pass_done = 1
    # movec 는 호를 따라가므로 실제 지난 거리는 현이 아니라 호 길이다.
    # 총 작업 거리는 TCP 가 실제로 움직인 길이다. EOAT 폭만큼 짧으므로
    # 덮는 길이(app_arc)가 아니라 arc_run 을 더한다.
    path_len = path_len + arc_run
    write_port_register(291, row_idx)
    pr2_w1(297, path_len * 0.1)
    pr2_w1(298, row_idx * 100.0 / rows)
      end
      $ LINE: (46, "If")
      if (row_idx<rows and dir_sign<0 and pass_done==0):
        $ LINE: (47, "8 [스크립트파일] dus_pass_l.script")
        $ LINE: (48, "스크립트")
    # =============================================================================
    #  dus_pass_l.script — dusan_v3
    #  왼쪽(Y-) 으로 한 줄. 중앙을 경유점으로 하는 movec 원호
    #
    #  펜던트에서 "8_pass_left" 자리에 스크립트 노드를 파일(File) 모드로 넣고 지정한다.
    #
    #  ※ def main() 으로 감싸지 말 것 (펜던트가 호출하지 않는다)
    #  ※ 최상위에 global 을 쓰지 말 것 (preamble 이 이미 선언·대입해 뒀다)
    #  ※ if / while 은 반드시 end 로 닫을 것
    # =============================================================================

    def pl2_w1(a, v):
      if (v > 32000):
        v = 32000
      end
      if (v < -32000):
        v = -32000
      end
      write_port_register(a, floor(v + 0.5))
    end


    # 왼쪽(Y-) 으로 한 줄 — movec 원호 하나
    z_now = get_actual_tcp_pose()[2]
    via_pose = p_c_pose.copy()
    via_pose[2] = z_now
    to_pose = zero_pose.copy()
    to_pose[2] = z_now
    movec(via_pose, to_pose, a = a_scan, v = v_scan, r = 0, mode = 1)

    row_idx = row_idx + 1
    dir_sign = 1
    pass_done = 1
    # movec 는 호를 따라가므로 실제 지난 거리는 현이 아니라 호 길이다.
    # 총 작업 거리는 TCP 가 실제로 움직인 길이다. EOAT 폭만큼 짧으므로
    # 덮는 길이(app_arc)가 아니라 arc_run 을 더한다.
    path_len = path_len + arc_run
    write_port_register(291, row_idx)
    pl2_w1(297, path_len * 0.1)
    pl2_w1(298, row_idx * 100.0 / rows)
      end
      $ LINE: (49, "If")
      if (row_idx<rows):
        $ LINE: (50, "9 [스크립트파일] dus_up.script")
        $ LINE: (51, "스크립트")
    # =============================================================================
    #  dus_up.script — dusan_v3
    #  다음 줄로 한 피치만큼 상승한다
    #
    #  펜던트에서 "9_up" 자리에 스크립트 노드를 파일(File) 모드로 넣고 지정한다.
    #
    #  ※ def main() 으로 감싸지 말 것 (펜던트가 호출하지 않는다)
    #  ※ 최상위에 global 을 쓰지 말 것 (preamble 이 이미 선언·대입해 뒀다)
    #  ※ if / while 은 반드시 end 로 닫을 것
    # =============================================================================

    def up_w1(a, v):
      if (v > 32000):
        v = 32000
      end
      if (v < -32000):
        v = -32000
      end
      write_port_register(a, floor(v + 0.5))
    end


    # 목표 높이는 직전 위치가 아니라 원점(z_base) 기준 절대값으로 잡는다.
    # 상대값으로 쌓으면 구간마다의 정지 오차가 행 수만큼 누적된다.
    tgt_pose = get_actual_tcp_pose()
    tgt_pose[2] = z_base + row_idx * pitch * 0.001
    movel(tgt_pose, a = a_scan, v = v_scan)

    path_len = path_len + pitch
    up_w1(297, path_len * 0.1)
      end
      $ LINE: (52, "If")
      if (row_idx>=rows):
        $ LINE: (53, "10 [스크립트파일] dus_finish.script")
        $ LINE: (54, "스크립트")
    # =============================================================================
    #  dus_finish.script — dusan_v3
    #  벽에서 후퇴하고 완료 플래그를 낸다
    #
    #  펜던트에서 "10_finish" 자리에 스크립트 노드를 파일(File) 모드로 넣고 지정한다.
    #
    #  ※ def main() 으로 감싸지 말 것 (펜던트가 호출하지 않는다)
    #  ※ 최상위에 global 을 쓰지 말 것 (preamble 이 이미 선언·대입해 뒀다)
    #  ※ if / while 은 반드시 end 로 닫을 것
    # =============================================================================

    tgt_pose = get_actual_tcp_pose()
    tgt_pose[0] = get_actual_tcp_pose()[0] - back_off * 0.001
    movel(tgt_pose, a = a_l, v = v_l)

    write_port_register(290, 5)
    write_port_register(291, row_idx)
    write_port_register(295, 1)
    write_port_register(298, 100)
        $ LINE: (55, "11 move_home")
        $ LINE: (56, "If")
        if (get_actual_tcp_pose()[2]<Home_pose[2]-0.001):
          $ LINE: (57, "MoveL")
          $ LINE: (58, "방향 로봇 Z+")
          global move_thread_flag_58
          move_thread_flag_58 = 0
          def move_thread_58():
            global move_thread_flag_58
            move_thread_flag_58 = 1
            towardsPos = calculate_point_to_move_towards([0.0, 0.0, 0.0, 0.0, 0.0, 0.0], [0.0,0.0,1.0], 1000.0)
            movel(towardsPos, a=0.6, v=0.15)
            move_thread_flag_58 = 2
          end
          move_thread_flag_58 = 0
          move_thread_han_58 = start_thread(move_thread_58, (), detach_mode = False)
          while (True):
            if (get_actual_tcp_pose()[2]>=Home_pose[2]-0.001):
              stop_thread(move_thread_han_58)
              stopl(0.6)
              $ LINE: (59, "Until (표현식)")
              break
            end
            sync()
          end
        end
        $ LINE: (60, "MoveJ")
        $ LINE: (61, "Home_joint", "after")
        movej(Home_joint, a=0.698131700835289, v=0.3490658503988659)
        $ LINE: (62, "중지")
        halt()
      end
      Loop_1 = Loop_1 + 1
    end
    $ LINE: (63, "중지")
    halt()
  end
end
